// TwinCAT 3 PLC project Simulator
// ProgramVersion: 3.1.4023.0
// libraries:
//   Tc2_Standard, * (Beckhoff Automation GmbH)
//   Tc2_System, * (Beckhoff Automation GmbH)
//   Tc2_Utilities, * (Beckhoff Automation GmbH)
//   Tc3_Module, * (Beckhoff Automation GmbH)
// project tree:
//   DUTs/ EachRecipeStep.TcDUT (not stored), Vessel.TcDUT
//   GVLs/ IO.TcGVL, R1.TcGVL
//   Helpers/ RemainingTimeCalculator.TcPOU (not stored), ShutDown.TcPOU (not stored), Simulator.TcPOU
//   / PlcTask.TcTTO (not stored)
//   POUs/ MAIN.TcPOU
//   RecipeModules/ InitializeRecipeModule.TcPOU (not stored), RecipeModule_R1.TcPOU (not stored)
// real-time tasks:
//   TASK PlcTask: cycle T#100000us, priority 20, ADS port 350

// ---- DUTs/Vessel.TcDUT
TYPE Vessel :
STRUCT
	LLS AT %I* : BOOL;	
	ULS AT %I* : BOOL;	
	
	VentValve AT %Q* : BOOL := FALSE;
	N2PurgeValve AT %Q* : BOOL := FALSE;
	TransferValve AT %Q* : BOOL := FALSE;
	FillInValve AT %Q* : BOOL := FALSE;
	FillInPump AT %Q* : BOOL := FALSE;
	TransferPump AT %Q* : BOOL := FALSE;
	FillInHeaderValve AT %Q* : BOOL := FALSE;

END_STRUCT
END_TYPE

// ---- GVLs/IO.TcGVL
{attribute 'qualified_only'}
VAR_GLOBAL
	R1 : Vessel;
	R2 : Vessel;
	R3 : Vessel;
	R4 : Vessel;
	R5 : Vessel;
END_VAR

// ---- GVLs/R1.TcGVL
VAR_GLOBAL

Test : DINT;
//****** VALVES *****//
	Valve_1 : BOOL;
	Valve_2 : BOOL;
	Valve_3 : BOOL;
	Valve_4 : BOOL;
	Valve_5 : BOOL;
	Valve_6 : BOOL;
	Valve_7 : BOOL;
	Valve_8 : BOOL;
	Valve_9 : BOOL;
	Valve_10 : BOOL;
	Valve_11 : BOOL;
	Valve_12 : BOOL;
	Valve_13 : BOOL;
	Valve_14 : BOOL;
	Valve_15 : BOOL;
	Valve_16 : BOOL;
	Valve_17 : BOOL;
	Valve_18 : BOOL;
	Valve_19 : BOOL;
	Valve_20 : BOOL;
	Valve_21 : BOOL;
	Valve_22 : BOOL;
	Valve_23 : BOOL;
	Valve_24 : BOOL;
	Valve_25 : BOOL;
	Valve_26 : BOOL;
	Valve_27 : BOOL;
	Valve_28 : BOOL;
	Valve_29 : BOOL;
	Valve_30 : BOOL;
	Valve_31 : BOOL;
	Valve_32 : BOOL;
	Valve_33 : BOOL;
	Valve_34 : BOOL;
	Valve_35 : BOOL;
	Valve_36 : BOOL;
	Valve_37 : BOOL;
	Valve_38 : BOOL;
	Valve_39 : BOOL;
	Valve_40 : BOOL;
	Valve_41 : BOOL;
	Valve_42 : BOOL;
	Valve_43 : BOOL;
	Valve_44 : BOOL;
	Valve_45 : BOOL;
	Valve_46 : BOOL;
	Valve_47 : BOOL;
	Valve_48 : BOOL;
	Valve_49 : BOOL;
	Valve_50 : BOOL;



//****** PUMPS *****//
	Pump_1 : BOOL;
	Pump_2 : BOOL;
	Pump_3 : BOOL;
	Pump_4 : BOOL;
	Pump_5 : BOOL;
	Pump_6 : BOOL;
	Pump_7 : BOOL;
	Pump_8 : BOOL;
	Pump_9 : BOOL;
	Pump_10 : BOOL;

	
//***** TAGS FOR HC ******//
	HeatCoolStatus : BOOL;
	HeatCoolSetPoint : DINT := 0;
	HeatCoolTemperatureControlType : BOOL; (* 0 - Jacket , 1 - Process *)
	HeatCoolStatusFeedback : BOOL;
	ReactorMassTemperature : REAL;
	JacketOutletTemperature : REAL;
	
// ***** TAGS FOR STIRRER *****//
	StirrerStatus : BOOL;
	StirrerStatusFeedback : BOOL;
	StirrerSetPoint : DINT;
	StirrerRPM : DINT;  (* Rotations Per Minute *)
	
// ***** TAGS FOR DOSING PUMP ******//
	DosingPumpStatus : BOOL;
	DosingPumpFlowSetPoint : REAL;
	DosingPumpFPM : REAL; (* Flow Per Minute *)
	DosingPumpStatusFeedback : BOOL;
	

//***** COMPULSORY UI TAGS *****//
	UsedNow : BOOL :=FALSE;
	EmergencyStatus :BOOL:=0;
	BatchText_1:STRING;
	BatchText_2:STRING;
	BatchText_3:STRING;
	BatchText_4:STRING;
	BatchText_5:STRING;


//****** TAGS FOR RECIPE ******//
	StepCount:INT:=0;
	TotalEnabledValue:INT:=0;
	TotalEndedValue:INT:=0;
	StepCompleted:BOOL:=0;
	NumberOfRecipeSteps : DINT := 0;
	RecipeStep: ARRAY[0..100] OF EachRecipeStep;
	RecipeStatus:BOOL:=0;
	ClearRecipe:BOOL:=0;
	AbortRecipe : BOOL := 0;
	RecipeEnded:BOOL;
	StartWaitTimer: BOOL; 
	DosingControlModeEmergency : BOOL;
	WaitTick:INT:=0;
	WaitSecondTick:INT:=0;
	WaitMinuteTick:INT:=0;
	ClearRecipeTrig:BOOL;
	 
END_VAR

// ---- Helpers/Simulator.TcPOU
FUNCTION_BLOCK Simulator
VAR_INPUT
	CurrentValue : REAL;
	TargetValue : REAL;
END_VAR
VAR_OUTPUT
	SimulatedValue : REAL;
END_VAR
VAR
	random_value : LREAL;
	fb_ran : DRAND;
END_VAR

fb_ran(Seed := 0, Num => random_value);
IF CurrentValue <= TargetValue THEN
	CurrentValue := CurrentValue + LREAL_TO_REAL(STRING_TO_LREAL(LREAL_TO_FMTSTR(random_value, 2, TRUE)));
ELSE
	CurrentValue := CurrentValue - LREAL_TO_REAL(STRING_TO_LREAL(LREAL_TO_FMTSTR(random_value, 2, TRUE)));
END_IF
SimulatedValue := STRING_TO_REAL(LREAL_TO_FMTSTR(CurrentValue, 2, TRUE)); //Rounding again here to clear any errors above

END_FUNCTION_BLOCK

// ---- POUs/MAIN.TcPOU
PROGRAM MAIN
VAR
	recipeInitializer : InitializeRecipeModule;
	fglocal : FB_LocalSystemTime;
	System_Time: TIMESTRUCT;
	currentHour : STRING;
	currentMinute : STRING;
	concatenatedHourMinuteString : STRING;
	
	ClearRecipeTrig_R1:R_Trig;
	NullRecipeStepArray : ARRAY[0..100] OF EachRecipeStep;
	
	CameraStatus : BOOL;
	LampStatus : BOOL;
	simulator : Simulator;
	random_value : REAL;
	
	timeCounter : INT;
	updateAllParameters : BOOL;
	skipCycleCounter : INT := 0;
END_VAR

IF updateAllParameters THEN
	//Update parameters for R1 using Simulator logic
	random_value := 0;
	simulator(CurrentValue := R1.JacketOutletTemperature, TargetValue := DINT_TO_REAL(R1.HeatCoolSetPoint), SimulatedValue => random_value);
	R1.JacketOutletTemperature := REAL_TO_INT(random_value);
	
	simulator(CurrentValue := R1.ReactorMassTemperature, TargetValue := R1.JacketOutletTemperature, SimulatedValue => random_value);
	R1.ReactorMassTemperature := random_value;
	
	random_value := 0;
	simulator(CurrentValue := DINT_TO_REAL(R1.StirrerRPM), TargetValue := DINT_TO_REAL(R1.StirrerSetPoint), SimulatedValue => random_value);
	R1.StirrerRPM := REAL_TO_INT(random_value);
	
	//Reset timeCounter
	updateAllParameters := FALSE;
	timeCounter := 0;
ELSE
	timeCounter := timeCounter + 1;
	IF timeCounter >= 5 THEN
		updateAllParameters := TRUE;
	END_IF
END_IF

recipeInitializer(GvlIdentifier := 1, ClearRecipe := R1.ClearRecipe);

END_PROGRAM
